{attribute 'qualified_only'}
VAR_GLOBAL
	fOutletFlow : LREAL := 0.0005;
END_VAR

(* stored: Version 1.1.0.1, ProductVersion 3.1.4024.10
   GVL Parameter: Id {43beea29-17be-44a1-825b-75a4ee47fe1e} *)
